{attribute 'qualified_only'}
{attribute 'strict'}
TYPE E_XMotion_Status :
(
	StartUp 	:= 0,
	Aborting 	:= 1,
	Aborted 	:= 2,	
	Resetting   := 3,
	Stopped  	:= 4,
	Preparing   := 5,
	Prepared    := 6,
	Execute 	:= 7,
	HoldOnError := 8
	
) DINT;
END_TYPE

(* stored: Version 1.1.0.1, ProductVersion 3.1.4024.5
   DUT E_XMotion_Status: Id {5ef50055-88a0-4666-b0c3-59fe08947d70} *)
